// TIA Portal V20 export
// export: Created 2025-12-01T14:57:10.8516778Z, ExportSetting None, DisplayName Totally Integrated Automation Portal, DisplayVersion V20 Update 3, DisplayName TIA Portal Openness, DisplayVersion V20 Update 3, DisplayName TIA Portal Version Control Interface, DisplayVersion V20 Update 3, DisplayName STEP 7 Professional, DisplayVersion V20 Update 3, DisplayName STEP 7 Safety, DisplayVersion V20 Update 2, DisplayName WinCC Basic/Comfort/Advanced, DisplayVersion V20 Update 3, DisplayName WinCC Professional, DisplayVersion V20 Update 3, DisplayName WinCC Unified, DisplayVersion V20 Update 3
FUNCTION "FC823_OrdenesMesas" : Void   // FC823, LAD
TITLE = "OrdenesMesas" - Calcular las ordenes de las UT's
{ S7_Optimized_Access := 'FALSE' }
AUTHOR : TRACKING
NAME : 20160407
VERSION : 4.1
// - Inicializaciones
// - Bucle de Mesas
// - Cierre del Protocolo de la Mesa 
// - Buscar Nueva Orden para enviar a la Mesa
// - Calacular la nueva Orden de la Mesa
// stored: AutoNumber false, SetENOAutomatically false
   VAR_TEMP
      RecProtocoloDeMesa : "UDT_ProtocoloRecMesa";
      P_RecProtocolo : DWord;
      P_Temporal : DWord;
      PLCOrden : Word;   // Estructura de recepcion de la mesa
      PLCOrdenAux_01 : UInt;   // Estructura de recepcion de la mesa (TipoCarga)
      PLCMesaSalidaMultiple : UInt;   // Estructura de recepcion de la mesa (Auxiliar 02)
      PLCOrdenAux_03 : UInt;   // Estructura de recepcion de la mesa (Auxiliar 03)
      PLCOrdenAux_04 : UInt;   // Estructura de recepcion de la mesa (Auxiliar 04)
      NumeroMesa : UInt;   // Numero de Mesa Actual
      NumeroUT : UInt;   // Numero de UT Actual
      SiguienteUT : UInt;   // Numero de UT Siguiente
      ValorReturn : Int;   // Temporal
   END_VAR
BEGIN

NETWORK
TITLE = Inicializar
// Inicializacion de las variables de los DB's
/////////////////////////////////////////////////////////////////////////
// Inicializaciones de las variables de los DB's

      L     0;
      T     #PLCOrden;
      T     #PLCMesaSalidaMultiple;
      T     #PLCOrdenAux_01;
      T     #PLCOrdenAux_03;
      T     #PLCOrdenAux_04;



NETWORK
TITLE = Bucle de Mesas
// - Inicializacion de variables de la mesa (PunteroMesa y PunteroPLC)
// - Mirar si ha cerrado el protocolo
/////////////////////////////////////////////////////////////////////////
/////////////////////////////////////////////////////////////////////////
/////////////////////////////////////////////////////////////////////////
// Inicializo variable, para bucle de mesas
      L     0;
      T     #NumeroMesa;


/////////////////////////////////////////////////////////////////////////
// Inicializo variable, para bucle de mesas
// Empieza el recorrido por todas las Mesas
InicioBucle_Mesas:NOP   0;
      L     #NumeroMesa;  // Incremento en uno el numero de mesa
      L     1;
      +I;
      T     #NumeroMesa;


/////////////////////////////////////////////////////////////////////////
// Ya he recorrido todas las Mesas
      L     #NumeroMesa;  // Ya estan todas las Mesas
      L     "CTE_MaxMesas";
      >I;
      JC    _END;


/////////////////////////////////////////////////////////////////////////
/// Mirar Si hay Mesa Configurada, No Definida no seguir
      SET;
      AN    "DB850_DefinicionMesas".Mesa[#NumeroMesa].ConfigMesa.MesaPaso;
      AN    "DB850_DefinicionMesas".Mesa[#NumeroMesa].ConfigMesa.MesaCruce;
      AN    "DB850_DefinicionMesas".Mesa[#NumeroMesa].ConfigMesa.MesaMultiplesDestinos;
      AN    "DB850_DefinicionMesas".Mesa[#NumeroMesa].ConfigMesa.MesaTL;
      JC    InicioBucle_Mesas;


/////////////////////////////////////////////////////////////////////////
/// Recoger Datos de Emision y Recepcion
      CALL  MOVE
      ( IN  := "DB841_Recepcion".Mesa[#NumeroMesa].Protocolo,
        OUT := #RecProtocoloDeMesa
      );

      L     P##RecProtocoloDeMesa;
      T     #P_RecProtocolo;

/////////////////////////////////////////////////////////////////////////
// Mirar si ha cerrado el protocolo de la Mesa de la anterior orden enviada

// --- 1º Condicion: Tiene que estar cerrado el protocolo
      L     "DB810_ColasMesas".Colas[#NumeroMesa].EstadoOrdenMesa;
      L     0;  // Mirar si no esta Cerrado el Protocolo
      <>I;  // Ir a Cerrar Protocolo de la Mesa
      JC    CerrarProtocolo_Mesa;


/////////////////////////////////////////////////////////////////////////
// Ir a Buscar Orden Nueva para la Mesa
      JU    TratarOrden_Mesa;



NETWORK
TITLE = Cierre del protocolo de la mesa
// - Recoger como esta el RecepOK
// - Distribuir dependiendo del Status del Protocolo
// - Esta en Fase 1 - Esperando que se desactive RecepOK de la Mesa
// - Esta en Fase 2 - Esperando que se active RecepOK de la Mesa
CerrarProtocolo_Mesa:NOP   0;

/////////////////////////////////////////////////////////////////////////
/////////////////////////////////////////////////////////////////////////
/////////////////////////////////////////////////////////////////////////
/////////////////////////////////////////////////////////////////////////
// Distribuir dependiendo del Status del protocolo

      L     "DB810_ColasMesas".Colas[#NumeroMesa].EstadoOrdenMesa;
      L     1;  // Protocolo - Esta en Fase 1
      ==I;
      JC    ProtocoloEnFase_01_Mesa;

// Protocolo - Esta en Fase 2
      JU    ProtocoloEnFase_02_Mesa;


/////////////////////////////////////////////////////////////////////////
/////////////////////////////////////////////////////////////////////////
// Esta en Fase 1 - Esperando que se desactive RecepOK de la Mesa
ProtocoloEnFase_01_Mesa:NOP   0;
      SET;  // Si esta 1 todavia no se puede dar pòr finalizado el protocolo
      A     "DB840_Emision".Mesa[#NumeroMesa].Protocolo.RecepOK;
      JC    FinCerrarProtocolo_Mesa;

// Pasar a Fase 0, Acabado el Protocolo
      L     0;  // Fase 0
      T     "DB810_ColasMesas".Colas[#NumeroMesa].EstadoOrdenMesa;

      JU    FinCerrarProtocolo_Mesa;


/////////////////////////////////////////////////////////////////////////
/////////////////////////////////////////////////////////////////////////
// Esta en Fase 2 - Esperando que se active RecepOK de la Mesa
ProtocoloEnFase_02_Mesa:NOP   0;
      SET;  // Si esta a 0 todavia no cambia a fase 1 el protocolo
      AN    "DB840_Emision".Mesa[#NumeroMesa].Protocolo.RecepOK;
      JC    FinCerrarProtocolo_Mesa;

// Pasar a Fase 1, Esperando que desactive el RecpOK
      L     LW [#P_RecProtocolo];
      L     W#16#80;  // Desactivo la Orden enviada todas menos el bit EmiOK
      AW;  // Y todos los Word Adicionales se ponen a 0
      T     LW [#P_RecProtocolo];  // Posicion - 8

      CALL  MOVE
      ( IN  := #RecProtocoloDeMesa,
        OUT := "DB841_Recepcion".Mesa[#NumeroMesa].Protocolo
      );

      L     0;  // Word Auxiliares
      T     "DB841_Recepcion".Mesa[#NumeroMesa].MesaSalidaMultiDestino;
      T     "DB841_Recepcion".Mesa[#NumeroMesa].Auxiliar_01;
      T     "DB841_Recepcion".Mesa[#NumeroMesa].Auxiliar_03;
      T     "DB841_Recepcion".Mesa[#NumeroMesa].Auxiliar_04;

      L     1;  // Fase 1
      T     "DB810_ColasMesas".Colas[#NumeroMesa].EstadoOrdenMesa;

      JU    FinCerrarProtocolo_Mesa;


/////////////////////////////////////////////////////////////////////////
/////////////////////////////////////////////////////////////////////////
// Final del Segmento del Cierre de Protocolo de la Mesa
FinCerrarProtocolo_Mesa:NOP   0;
// Finalizar, ir a la siguiente Mesa
      JU    InicioBucle_Mesas;



NETWORK
TITLE = Buscar Nueva Orden a enviar al PLC (Solo la primera UT)
// - Mirar is hay UT (Solo tiene que enviar la primera de cada mesa)
// - Mirar como esta el VI (Estado)
// - Mirar si esta todo Emitido
// - Mirar si ha cambiado de Mesa
// - Mirar si ha recibido Evento
TratarOrden_Mesa:NOP   0;
      L     0;
      T     #PLCOrden;
      T     #PLCMesaSalidaMultiple;
      T     #PLCOrdenAux_01;
      T     #PLCOrdenAux_03;
      T     #PLCOrdenAux_04;

/////////////////////////////////////////////////////////////////////////
/////////////////////////////////////////////////////////////////////////
/////////////////////////////////////////////////////////////////////////
      L     "DB810_ColasMesas".Colas[#NumeroMesa].UT_PrimeraMesa;
      T     #NumeroUT;

/////////////////////////////////////////////////////////////////////////
// --- Mirar si hay UT, Si hay Inicializo el Puntero
// --- 1º Condicion: Tiene que haber UT en la Mesa

      L     #NumeroUT;  // Mirar si hay UT ?
      L     0;
      ==I;  // No hay UT
      JC    FinTratarOrden_Mesa;


/////////////////////////////////////////////////////////////////////////
// --- 2º Condicion: El estado del VI  ¡¡¡ ANALIZAR !!!
// ---   ¿Mirar como esta el VI?
// ---   ¿Solo cuando esta en Carga o reposo?
// ---   ¿Da lo mismo, menos en Reset?


/////////////////////////////////////////////////////////////////////////
// --- 3º Condicion: Estado del Dispositivo
// --- Condición >>> Marcha + Auto (EmisionDeDispositivoMesa)
// Marcha + Auto >> Sino esta asi NO puede Calcular la orden
      SET;
      A     "DB840_Emision".DispoMesa[#NumeroMesa].Protocolo.Automatico;
      A     "DB840_Emision".DispoMesa[#NumeroMesa].Protocolo.Marcha;
      JCN   FinTratarOrden_Mesa;


/////////////////////////////////////////////////////////////////////////
// --- Mirar si esta todo Emitido (StatusEmisionUT = 0)
// --- 4º Condicion: La UT no tiene nada Evento que Generar
//                   (Lo logico es que este libre, menos en un reset)
      L     "DB812_UTs_Control".UT[#NumeroUT].EstadoEmisionUT;
      L     0;
      <>I;  // Esta emitido todo ?
      JC    FinTratarOrden_Mesa;


/////////////////////////////////////////////////////////////////////////
/////////////////////////////////////////////////////////////////////////
/////////////////////////////////////////////////////////////////////////
// --- Mirar Si ha cambiado de estado (StatatusRecepcionUT <> 0)
// --- 1º Caso para el Calculo de Orden: Nueva UT ó Cambia Mesa
      L     "DB812_UTs_Control".UT[#NumeroUT].EstadoRecepcionUT;
      L     0;
      <>I;  // Si tiene para enviar orden ?
      JC    CalcularOrden_FASE01_Mesa;


/////////////////////////////////////////////////////////////////////////
/////////////////////////////////////////////////////////////////////////
/////////////////////////////////////////////////////////////////////////
// --- Mirar si ha Recibido Eventos (StatatusEventoRecibido <> 0)
// --- 2º Caso para el Calculo de Orden: Evento Recibido
// --- (Hay eventos que no tienen)
      L     "DB812_UTs_Control".UT[#NumeroUT].EstadoEventoRecibido;
      L     0;
      <>I;  // Si ha recibido Evento ?
      JC    RecibidoEvento_Mesa;


/////////////////////////////////////////////////////////////////////////
/////////////////////////////////////////////////////////////////////////
/////////////////////////////////////////////////////////////////////////
// No esta, no se puede enviar nada
      JU    FinTratarOrden_Mesa;


/////////////////////////////////////////////////////////////////////////
/////////////////////////////////////////////////////////////////////////
/////////////////////////////////////////////////////////////////////////
// Final del Segmento de Buscar Nueva Orden a enviar al PLC
FinTratarOrden_Mesa:NOP   0;
// Finalizar, ir a la siguiente Mesa
      JU    InicioBucle_Mesas;



NETWORK
TITLE = Recibido Evento para la Mesa
// - Distribucion dependiendo del ento recibido
// - Eventos que no necesitan Orden
//     - Recibido Evento de Borrar UT
//     - Recibido Evento de Refresco de datos la UT
// 
// -Eventos que puede ser que necesite orden
//     - Recibido Evento de Ruta Nueva
//     - Recibido Evento de Nueva UT Creada
//     - Recibido Evento de Nuevos Datos para la UT
//     - Recibido Evento de Retirar la UT
RecibidoEvento_Mesa:NOP   0;

/////////////////////////////////////////////////////////////////////////
/////////////////////////////////////////////////////////////////////////
/////////////////////////////////////////////////////////////////////////
// Distribucion de los Eventos Recibidos

      L     "DB812_UTs_Control".UT[#NumeroUT].EstadoEventoRecibido;
      L     201;  // 201 - Ruta Nueva
      ==I;
      JC    EventoRecido_RutaNuevaUT_Mesa;

      L     "DB812_UTs_Control".UT[#NumeroUT].EstadoEventoRecibido;
      L     202;  // 202 - UT Creada
      ==I;
      JC    EventoRecido_CreadaUT_Mesa;

      L     "DB812_UTs_Control".UT[#NumeroUT].EstadoEventoRecibido;
      L     203;  // 203 - BorrarUT
      ==I;
      JC    EventoRecido_BorrarUT_Mesa;

      L     "DB812_UTs_Control".UT[#NumeroUT].EstadoEventoRecibido;
      L     204;  // 204 - Datos Nuevos de la UT
      ==I;
      JC    EventoRecido_DatosNuevosUT_Mesa;

      L     "DB812_UTs_Control".UT[#NumeroUT].EstadoEventoRecibido;
      L     205;  // 205 - Referesco de Datos
      ==I;
      JC    EventoRecido_RefrescoDatosUT_Mesa;


/////////////////////////////////////////////////////////////////////////
// --- Solo queda este tipo de evento: Retirar UT
      L     "DB812_UTs_Control".UT[#NumeroUT].EstadoEventoRecibido;
      L     210;  // 210...214 - Retirar UT
      <I;  // < 210 ? - No es Retirar UT
      JC    NoRecibidoEvento_Retirar_Mesa;
      L     "DB812_UTs_Control".UT[#NumeroUT].EstadoEventoRecibido;
      L     214;  // 210...214 - Retirar UT
      >I;  // > 214 ? - No es Retirar UT
      JC    NoRecibidoEvento_Retirar_Mesa;

      SET;  // Si es orden de Retirar UT (Simple)
      AN    "DB850_DefinicionMesas".Mesa[#NumeroMesa].ConfigMesa.AusenciaMultiple;
      JC    EventoRecido_RetiradaSimpleUT_Mesa;

// Si es orden de Retirar UT (Multiple)
      JU    EventoRecido_RetiradaMultipleUT_Mesa;

NoRecibidoEvento_Retirar_Mesa:NOP   0;


/////////////////////////////////////////////////////////////////////////
// --- El evento recibido no lo espera el sistema  ¡¡¡ MALO, MALO, MALO !!!

      L     0;  // Dar por tratado el Evento
      L     "DB812_UTs_Control".UT[#NumeroUT].EstadoEventoRecibido;


// Fin del Tratamiento del Eventos
      JU    FinRecibidoEvento_Mesa;


/////////////////////////////////////////////////////////////////////////
/////////////////////////////////////////////////////////////////////////
/////////////////////////////////////////////////////////////////////////
/////////////////////////////////////////////////////////////////////////
// --- Final de tratamiento de los Eventos Recibidos
FinRecibidoEvento_Mesa:NOP   0;
// Finalizar, ir a la siguiente Mesa
      JU    InicioBucle_Mesas;



NETWORK
TITLE = --- Lista de Eventos Recibidos
/////////////////////////////////////////////////////////////////////////
/////////////////////////////////////////////////////////////////////////
/////////////////////////////////////////////////////////////////////////
//
//                  LISTA DE EVENTOS QUE SE PUEDEN RECIBIR
//                        QUE HACER EN CADA CASO
//
/////////////////////////////////////////////////////////////////////////
/////////////////////////////////////////////////////////////////////////
/////////////////////////////////////////////////////////////////////////


/////////////////////////////////////////////////////////////////////////
/////////////////////////////////////////////////////////////////////////
// --- Evento que no necesita Orden
// 203 --- Recibido Evento de Borrar _UT
EventoRecido_BorrarUT_Mesa:NOP   0;
      L     "DB812_UTs_Control".UT[#NumeroUT].EstadoGeneralUT;
      L     0;  // Si EstadoGeneralUT = 0
      <>I;  // Esta Libre ?
      JC    FinRecibidoEvento_Mesa;


// Continuar con el ciclo
      L     0;  // Dar por tratado el Evento
      T     "DB812_UTs_Control".UT[#NumeroUT].EstadoEventoRecibido;
      L     31;  // 31 - Peticion de Borrado de UT
      T     "DB812_UTs_Control".UT[#NumeroUT].EstadoGeneralUT;


// Fin del Tratamiento del Evento
      JU    FinRecibidoEvento_Mesa;


/////////////////////////////////////////////////////////////////////////
/////////////////////////////////////////////////////////////////////////
// --- Evento que no necesita Orden
// 205 --- Recibido Evento de Refresco de Datos de la UT
EventoRecido_RefrescoDatosUT_Mesa:NOP   0;
      L     "DB812_UTs_Control".UT[#NumeroUT].EstadoGeneralUT;  // EstadoGeneralUT = 0
      L     0;
      <>I;
      JC    FinRecibidoEvento_Mesa;  // Esta Libre ?


// Continuar con el ciclo
      L     0;  // Dar por tratado el Evento
      T     "DB812_UTs_Control".UT[#NumeroUT].EstadoEventoRecibido;
      L     22;  // 22 - Peticion de Refresco de datos
      T     "DB812_UTs_Control".UT[#NumeroUT].EstadoGeneralUT;


// Fin del Tratamiento del Evento
      JU    FinRecibidoEvento_Mesa;




/////////////////////////////////////////////////////////////////////////
/////////////////////////////////////////////////////////////////////////
/////////////////////////////////////////////////////////////////////////
/////////////////////////////////////////////////////////////////////////
// --- Evento que puede ser que necesite Orden
// 201 --- Recibido Evento de Ruta Nueva
EventoRecido_RutaNuevaUT_Mesa:NOP   0;
      L     0;  // Dar por tratado el Evento
      T     "DB812_UTs_Control".UT[#NumeroUT].EstadoEventoRecibido;
      L     17;  // 17 - Ruta Nueva
      T     "DB812_UTs_Control".UT[#NumeroUT].EstadoRecepcionUT;


// Ir a calcular la Nueva Orden
      JU    CalcularOrden_FASE01_Mesa;


/////////////////////////////////////////////////////////////////////////
/////////////////////////////////////////////////////////////////////////
// --- Evento que puede ser que necesite Orden
// 202 --- Recibido Evento de Nueva UT Creada
EventoRecido_CreadaUT_Mesa:NOP   0;
      L     0;  // Dar por tratado el Evento
      T     "DB812_UTs_Control".UT[#NumeroUT].EstadoEventoRecibido;
      L     16;  // 16 - UT Creada
      T     "DB812_UTs_Control".UT[#NumeroUT].EstadoRecepcionUT;


// Ir a calcular la Nueva Orden
      JU    CalcularOrden_FASE01_Mesa;


/////////////////////////////////////////////////////////////////////////
/////////////////////////////////////////////////////////////////////////
// --- Evento que puede ser que necesite Orden
// 204 --- Recibido Evento de Nuevos datos de la UT
EventoRecido_DatosNuevosUT_Mesa:NOP   0;
      L     0;  // Dar por tratado el Evento
      T     "DB812_UTs_Control".UT[#NumeroUT].EstadoEventoRecibido;
      L     15;  // 15 - Nuevos Datos de UT
      T     "DB812_UTs_Control".UT[#NumeroUT].EstadoRecepcionUT;


// Ir a calcular la Nueva Orden
      JU    CalcularOrden_FASE01_Mesa;



NETWORK
TITLE = --- Evento Recibido de Retirada (Control Especial)
/////////////////////////////////////////////////////////////////////////
/////////////////////////////////////////////////////////////////////////
// --- Evento que puede ser que necesite Orden (Simple)
// 210... 214 --- Recibido Evento de Retirar UT de la mesa
EventoRecido_RetiradaSimpleUT_Mesa:NOP   0;

// Activar Bit Recibido del Evento
      L     P##PLCOrden;  // Dirección de la Orden del PLC
      T     #P_Temporal;

      L     "DB812_UTs_Control".UT[#NumeroUT].EstadoEventoRecibido;
      L     210;
      -I;  // Numero de Bit a Activar
      L     #P_Temporal;
      +D;
      T     #P_Temporal;  // Direccion del Bit a Activar

      SET;  // Poner a '1' el bit de la orden
      S     L [#P_Temporal];  // Orden del PLC calculada


// Finalizar Evento Recibido
      L     0;  // Dar por tratado el Evento
      T     "DB812_UTs_Control".UT[#NumeroUT].EstadoEventoRecibido;


/////////////////////////////////////////////////////////////////////////
// Enviar la Orden al PLC
      JU    EnviarOrden_Al_PLC;




/////////////////////////////////////////////////////////////////////////
/////////////////////////////////////////////////////////////////////////
// --- Evento que puede ser que necesite Orden (Multiple)
// 210... 214 --- Recibido Evento de Retirar UT de la mesa
EventoRecido_RetiradaMultipleUT_Mesa:NOP   0;

      L     "DB812_UTs_Control".UT[#NumeroUT].UT_SiguienteMesa;
      T     #SiguienteUT;

/////////////////////////////////////////////////////////////////////////
// --- Primero Mirar si ha llegado la orden de Retirar a todas las UT's
InicioBucleVerificar_RetiradaMultipleUT_Mesa:NOP   0;
      L     #SiguienteUT;
      L     0;  // No hay más UT's
      ==I;  // No hay más UT's enviar Retirar
      JC    FinBucleVerificar_RetiradaMultipleUT_Mesa;

// EventoRecibido de la Primera UT == Evento Recibido de todas las UTs
      L     "DB812_UTs_Control".UT[#SiguienteUT].EstadoEventoRecibido;
      L     "DB812_UTs_Control".UT[#NumeroUT].EstadoEventoRecibido;
      <>I;  // Tienen que ser iguales todas las UTs
      JC    FinRecibidoEvento_Mesa;

// Recorrer todas las UT's
      L     "DB812_UTs_Control".UT[#SiguienteUT].UT_SiguienteMesa;
      T     #SiguienteUT;

      JU    InicioBucleVerificar_RetiradaMultipleUT_Mesa;

// Final de Veficacion, Todas las Uts tienen Retirada
FinBucleVerificar_RetiradaMultipleUT_Mesa:NOP   0;


/////////////////////////////////////////////////////////////////////////
// Activar Bit Recibido del Evento
      L     P##PLCOrden;  // Dirección de la Orden del PLC
      T     #P_Temporal;

      L     "DB812_UTs_Control".UT[#NumeroUT].EstadoEventoRecibido;
      L     210;
      -I;  // Numero de Bit a Activar
      L     #P_Temporal;
      +D;
      T     #P_Temporal;  // Direccion del Bit a Activar

      SET;  // Poner a '1' el bit de la orden
      S     L [#P_Temporal];  // Orden del PLC calculada


/////////////////////////////////////////////////////////////////////////
// Dar por tratado el Evento Recibido Primera UT
      L     0;  // Dar por tratado el Evento
      T     "DB812_UTs_Control".UT[#NumeroUT].EstadoEventoRecibido;


/////////////////////////////////////////////////////////////////////////
// Dar por tratado el Evento Recibido al Resto de UT's
      L     "DB812_UTs_Control".UT[#NumeroUT].UT_SiguienteMesa;
      T     #SiguienteUT;

InicioBucleTratado_RetiradaMultipleUT_Mesa:NOP   0;
      L     #SiguienteUT;
      L     0;  // No hay más UT's
      ==I;  // No hay más UT's Finalizado
      JC    FinBucleTratado_RetiradaMultipleUT_Mesa;

// Dar por tratado el Evento
      L     0;  // Dar por tratado el Evento
      T     "DB812_UTs_Control".UT[#SiguienteUT].EstadoEventoRecibido;

// Recorrer todas las UT's
      L     "DB812_UTs_Control".UT[#SiguienteUT].UT_SiguienteMesa;
      T     #SiguienteUT;

      JU    InicioBucleTratado_RetiradaMultipleUT_Mesa;

// Final de Tratado, Todas las Uts tienen tratado el Evenfo
FinBucleTratado_RetiradaMultipleUT_Mesa:NOP   0;


/////////////////////////////////////////////////////////////////////////
/////////////////////////////////////////////////////////////////////////
// Enviar la Orden al PLC
      JU    EnviarOrden_Al_PLC;




NETWORK
TITLE = Calcular Orden - FASE 01 (Distribucion Causa) ---- Nota >>> Primera UT de la Mesa
CalcularOrden_FASE01_Mesa:NOP   0;

/////////////////////////////////////////////////////////////////////////
/////////////////////////////////////////////////////////////////////////
/////////////////////////////////////////////////////////////////////////
// Distribucion segun la causa:

      L     "DB812_UTs_Control".UT[#NumeroUT].EstadoRecepcionUT;
      L     11;  //  - (11) : Cambiado de Mesa la UT
      ==I;
      JC    CambiadaDeMesa_CalcularOrden_Mesa;

      L     "DB812_UTs_Control".UT[#NumeroUT].EstadoRecepcionUT;
      L     12;  //  - (12) : Nueva UT en Mesa
      ==I;
      JC    NuevaEnMesa_CalcularOrden_Mesa;

      L     "DB812_UTs_Control".UT[#NumeroUT].EstadoRecepcionUT;
      L     13;  //  - (13) : Reset del PLC
      ==I;
      JC    ResetEnMesa_CalcularOrden_Mesa;

      L     "DB812_UTs_Control".UT[#NumeroUT].EstadoRecepcionUT;
      L     15;  //  - (15) : Datos Nuevos de la UT
      ==I;
      JC    DatosNuevos_CalcularOrden_Mesa;

      L     "DB812_UTs_Control".UT[#NumeroUT].EstadoRecepcionUT;
      L     16;  //  - (16) : Creada UT
      ==I;
      JC    CreadaEnMesa_CalcularOrden_Mesa;

      L     "DB812_UTs_Control".UT[#NumeroUT].EstadoRecepcionUT;
      L     17;  //  - (17) : Recibida Nueva Ruta para la UT
      ==I;
      JC    RutaNueva_CalcularOrden_Mesa;


/////////////////////////////////////////////////////////////////////////
// --- No es una causa programada (Darla por tradada)
      L     0;  // Dar por tratada
      T     "DB812_UTs_Control".UT[#NumeroUT].EstadoRecepcionUT;

// No hay más que hacer
      JU    InicioBucle_Mesas;



NETWORK
TITLE = --- EstadoRecepcion (11) : Cambiado de Mesa la UT
// Pasos a Seguir: 
// - Mirar condiciones que debe cumplir
// - Calcular la Orden a Enviar
// - Darla por tratada y enviar la orden si es necesario
CambiadaDeMesa_CalcularOrden_Mesa:NOP   0;

/////////////////////////////////////////////////////////////////////////
/////////////////////////////////////////////////////////////////////////
/////////////////////////////////////////////////////////////////////////
// (11) : Cambiado de Mesa la UT


/////////////////////////////////////////////////////////////////////////
// --- Mirar condiciones que debe cumplir


/////////////////////////////////////////////////////////////////////////
// --- Calcular Orden
      JU    CalcularOrden_FASE02_Mesa;



NETWORK
TITLE = --- EstadoRecepcion (12) : Nueva UT en Mesa
// Pasos a Seguir: 
// - Mirar condiciones que debe cumplir
// - Calcular la Orden a Enviar
// - Darla por tratada y enviar la orden si es necesario
NuevaEnMesa_CalcularOrden_Mesa:NOP   0;

/////////////////////////////////////////////////////////////////////////
/////////////////////////////////////////////////////////////////////////
/////////////////////////////////////////////////////////////////////////
// (12) : Nueva UT en Mesa


/////////////////////////////////////////////////////////////////////////
// --- Mirar condiciones que debe cumplir


/////////////////////////////////////////////////////////////////////////
// --- Se da la causa por tratata, no se envia orden
      L     0;  // Dar por tratada
      T     "DB812_UTs_Control".UT[#NumeroUT].EstadoRecepcionUT;

// No hay más que hacer
      JU    InicioBucle_Mesas;



NETWORK
TITLE = --- EstadoRecepcion (13) : Reset de la UT
// Pasos a Seguir: 
// - Mirar condiciones que debe cumplir
// - Calcular la Orden a Enviar
// - Darla por tratada y enviar la orden si es necesario
ResetEnMesa_CalcularOrden_Mesa:NOP   0;

/////////////////////////////////////////////////////////////////////////
/////////////////////////////////////////////////////////////////////////
/////////////////////////////////////////////////////////////////////////
// (13) : Reset de la UT

/////////////////////////////////////////////////////////////////////////
// --- Mirar condiciones que debe cumplir


/////////////////////////////////////////////////////////////////////////
// --- Calcular Orden
      JU    CalcularOrden_FASE02_Mesa;



NETWORK
TITLE = --- EstadoRecepcion (15) : Datos Nuevos de la UT
// Pasos a Seguir: 
// - Mirar condiciones que debe cumplir
// - Calcular la Orden a Enviar
// - Darla por tratada y enviar la orden si es necesario
DatosNuevos_CalcularOrden_Mesa:NOP   0;

/////////////////////////////////////////////////////////////////////////
/////////////////////////////////////////////////////////////////////////
/////////////////////////////////////////////////////////////////////////
// (15) : Datos Nuevos de la UT


/////////////////////////////////////////////////////////////////////////
// --- Mirar condiciones que debe cumplir


/////////////////////////////////////////////////////////////////////////
// --- Se da la causa por tratata, no se envia orden
      L     0;  // Dar por tratada
      T     "DB812_UTs_Control".UT[#NumeroUT].EstadoRecepcionUT;

// No hay más que hacer
      JU    InicioBucle_Mesas;



NETWORK
TITLE = --- EstadoRecepcion (16) : Creada UT
// Pasos a Seguir: 
// - Mirar condiciones que debe cumplir
// - Calcular la Orden a Enviar
// - Darla por tratada y enviar la orden si es necesario
CreadaEnMesa_CalcularOrden_Mesa:NOP   0;

/////////////////////////////////////////////////////////////////////////
/////////////////////////////////////////////////////////////////////////
/////////////////////////////////////////////////////////////////////////
// (16) : Creada UT


/////////////////////////////////////////////////////////////////////////
// --- Mirar condiciones que debe cumplir


/////////////////////////////////////////////////////////////////////////
// --- Se da la causa por tratata, no se envia orden
      L     0;  // Dar por tratada
      T     "DB812_UTs_Control".UT[#NumeroUT].EstadoRecepcionUT;

// No hay más que hacer
      JU    InicioBucle_Mesas;



NETWORK
TITLE = --- EstadoRecepcion (17) : Recibida Nueva Ruta para la UT
// Pasos a Seguir: 
// - Mirar condiciones que debe cumplir
// - Calcular la Orden a Enviar
// - Darla por tratada y enviar la orden si es necesario
RutaNueva_CalcularOrden_Mesa:NOP   0;

/////////////////////////////////////////////////////////////////////////
/////////////////////////////////////////////////////////////////////////
/////////////////////////////////////////////////////////////////////////
// (17) : Recibida Nueva Ruta para la UT


/////////////////////////////////////////////////////////////////////////
// --- Mirar condiciones que debe cumplir


/////////////////////////////////////////////////////////////////////////
// --- Calcular Orden
      JU    CalcularOrden_FASE02_Mesa;



NETWORK
TITLE = Calcular Orden - FASE 02 (Control Comun de la UT)
CalcularOrden_FASE02_Mesa:NOP   0;

/////////////////////////////////////////////////////////////////////////
/////////////////////////////////////////////////////////////////////////
/////////////////////////////////////////////////////////////////////////
//                    OPERATIVA NORMAL DE FUNCIONAMIENTO
/////////////////////////////////////////////////////////////////////////
// Casos que se puede dar:
//
// 1 Si no tiene Mckey, No debe darse este caso, tenerlo previsto.
//   Realizar, Evento de Nueva UT en Mesa (NUNCA SE DARA)
// 2 Sino tiene Ruta, MesaDestino = 0 (NUNCA SE DARA)
//   Realizar, Evento de Pedir Nueva Ruta
// 3 Si tiene ruta y ha llegado a su destino
// 4 Si tiene ruta y no ha llegado a su destino
//
/////////////////////////////////////////////////////////////////////////


/////////////////////////////////////////////////////////////////////////
// --- 1º Caso: El Mckey = 0 (Evento de Nueva UT en Mesa)
/////////////////////////////////////////////////////////////////////////
// El McKey = 0 (Evento de Nueva UT en la Mesa)
// Este caso NUNCA se dará, pero se programa por si acaso.
      SET;
      L     "DB812_UTs_Control".UT[#NumeroUT].Mckey;
      L     0;
      ==D;  // Tiene Mckey ?
      JC    NoEsxiteMckey_CalcularOrden_Mesa;


/////////////////////////////////////////////////////////////////////////
// --- 2º Caso: No tiene Ruta (MesaDestino = 0) (Evento de Pedir Ruta)
/////////////////////////////////////////////////////////////////////////
// El MesaDestino = 0 (Evento de Pedir Ruta Nueva)
// Este caso NUNCA se dará, pero se programa por si acaso.

      SET;  // Memoria de Recibido la Orden RETI (Prioritario)
      A     "DB812_UTs_Control".UT[#NumeroUT].AtributosDeLaUT.MemorizarRETI;
      JC    MemorizadoRetirada_CalcularOrden_Mesa;

      L     "DB812_UTs_Control".UT[#NumeroUT].MesaDestino;
      L     0;  // No tiene destino
      ==I;  // Tiene Ruta ?
      JC    SinDestino_CalcularOrden_Mesa;


/////////////////////////////////////////////////////////////////////////
// --- 3º Caso: Hay Ruta, y ha llegado a su destino (MesaDestino = MesaActual)
// --- MODIFICACION 06/05/2013 --> Recircular Activado, debe dar una vuelta completa
// ---       Aunque ha llegado su Destino, si esta activado la Marca
// ---       debe recircular siempre.

      SET;  // Memoria de Recibido la Orden RETI (Prioritario)
      A     "DB812_UTs_Control".UT[#NumeroUT].AtributosDeLaUT.MemorizarRETI;
      JC    MemorizadoRetirada_CalcularOrden_Mesa;

      SET;  // Solo para mesas de Cruce, Debe Recicular
      A     "DB812_UTs_Control".UT[#NumeroUT].AtributosDeLaUT.RecircularCarga;
      A     "DB850_DefinicionMesas".Mesa[#NumeroMesa].ConfigMesa.MesaCruce;
      JC    NoComprobarDestino_CalcularOrden_Mesa;

      L     "DB812_UTs_Control".UT[#NumeroUT].MesaDestino;
      L     "DB812_UTs_Control".UT[#NumeroUT].MesaActual;
      ==I;  // Ha llegado a su Destino ?
      JC    EnDestino_CalcularOrden_Mesa;

// Fin de Control de Llegada a Destino
NoComprobarDestino_CalcularOrden_Mesa:NOP   0;


/////////////////////////////////////////////////////////////////////////
// --- 4º Caso: Hay Ruta, y no ha llegado a su destino (MesaDestino <> MesaActual)
//     La UT esta de camino a su destino, dependiendo del tipo de mesa


/////////////////////////////////////////////////////////////////////////
// --- Si Bit de la Definicion de la Mesa "EspecialOrdenes", Hay funcion especial
//     que calcula la orden a enviar

      SET;
      A     "DB850_DefinicionMesas".Mesa[#NumeroMesa].ConfigMesa.EspecialOrdenes;  // Hay funcion particular
      JC    InicioBucle_Mesas;  // Aqui no hay nada que hacer


/////////////////////////////////////////////////////////////////////////
// --- Hay que hacer cosas diferentes, dependiendo del Tipo de Mesa:
//     * Mesa tipo de PASO
//     * Mesa tipo de CRUCE
//     * Mesa tipo de MUTIPLES DESTINOS
//     * Si no hay definido >>> No se Hace Nada

      SET;  // Es una Mesa de Paso
      A     "DB850_DefinicionMesas".Mesa[#NumeroMesa].ConfigMesa.MesaPaso;
      JC    MesaDePaso_CalcularOrden_Mesa;

      SET;  // Es una Mesa de Cruce
      A     "DB850_DefinicionMesas".Mesa[#NumeroMesa].ConfigMesa.MesaCruce;
      JC    MesaDeCruce_CalcularOrden_Mesa;

      SET;  // Es una Mesa de Multiples Destinos
      A     "DB850_DefinicionMesas".Mesa[#NumeroMesa].ConfigMesa.MesaMultiplesDestinos;
      JC    MesaDeMultiplesDestinos_CalcularOrden_Mesa;


/////////////////////////////////////////////////////////////////////////
// Tienen que estar la MESA configurada
      JU    InicioBucle_Mesas;



NETWORK
TITLE = --- Control (CASO) : No Tiene Mckey
NoEsxiteMckey_CalcularOrden_Mesa:NOP   0;

/////////////////////////////////////////////////////////////////////////
/////////////////////////////////////////////////////////////////////////
/////////////////////////////////////////////////////////////////////////
/////////////////////////////////////////////////////////////////////////
// --- El Mckey = 0 (Evento de Nueva UT en Mesa)
/////////////////////////////////////////////////////////////////////////
// El McKey = 0 (Evento de Nueva UT en la Mesa)
// Este caso NUNCA se dará, pero se programa por si acaso.


/////////////////////////////////////////////////////////////////////////
// Condiciones -- EstadoGeneralUT = 0
      L     "DB812_UTs_Control".UT[#NumeroUT].EstadoGeneralUT;
      L     0;  // Libre
      <>I;  // NO esta LIBRE ?
      JC    InicioBucle_Mesas;


/////////////////////////////////////////////////////////////////////////
// Acciones:   -- EstadoGeneralUT = 24 (Evento de Nueva UT en Mesa)
//             -- EstadoRecepcionUT = 0
      L     24;  // 24 - Generar Evento Nueva UT en Mesa
      T     "DB812_UTs_Control".UT[#NumeroUT].EstadoGeneralUT;
      L     0;  // Dar por tratada
      T     "DB812_UTs_Control".UT[#NumeroUT].EstadoRecepcionUT;

// No hay más que hacer
      JU    InicioBucle_Mesas;



NETWORK
TITLE = --- Control (CASO) : No tiene Destino
SinDestino_CalcularOrden_Mesa:NOP   0;

/////////////////////////////////////////////////////////////////////////
/////////////////////////////////////////////////////////////////////////
/////////////////////////////////////////////////////////////////////////
/////////////////////////////////////////////////////////////////////////
// --- No tiene Ruta (MesaDestino = 0) (Evento de Pedir Ruta)
/////////////////////////////////////////////////////////////////////////
// El MesaDestino = 0 (Evento de Pedir Ruta Nueva)
// Este caso NUNCA se dará, pero se programa por si acaso.


/////////////////////////////////////////////////////////////////////////
// Condiciones -- EstadoGeneralUT = 0
      L     "DB812_UTs_Control".UT[#NumeroUT].EstadoGeneralUT;
      L     0;  // Libre
      <>I;  // NO esta LIBRE ?
      JC    InicioBucle_Mesas;


/////////////////////////////////////////////////////////////////////////
// Acciones:   -- EstadoGeneralUT = 25 (Evento de Pedir Ruta Nueva)
//             -- EstadoRecepcionUT = 0
      L     25;  // 25 - Generar Evento Pedir Ruta (SIN DESTINO)
      T     "DB812_UTs_Control".UT[#NumeroUT].EstadoGeneralUT;
      L     0;  // Dar por tratada
      T     "DB812_UTs_Control".UT[#NumeroUT].EstadoRecepcionUT;

// No hay más que hacer
      JU    InicioBucle_Mesas;



NETWORK
TITLE = --- Control (CASO) : En Destino
EnDestino_CalcularOrden_Mesa:NOP   0;

/////////////////////////////////////////////////////////////////////////
/////////////////////////////////////////////////////////////////////////
/////////////////////////////////////////////////////////////////////////
/////////////////////////////////////////////////////////////////////////
// --- Ha llegado a su desetino (Evento de Pedir Ruta)
/////////////////////////////////////////////////////////////////////////
// MesaActual = MesaDestino(Evento de Pedir Ruta Nueva)


/////////////////////////////////////////////////////////////////////////
// Condiciones -- EstadoGeneralUT = 0
      L     "DB812_UTs_Control".UT[#NumeroUT].EstadoGeneralUT;
      L     0;  // Libre
      <>I;  // NO esta LIBRE ?
      JC    InicioBucle_Mesas;


/////////////////////////////////////////////////////////////////////////
// Acciones:   -- EstadoGeneralUT = 21 (Evento de Pedir Ruta Nueva)
//             -- EstadoRecepcionUT = 0
      L     21;  // 21 - Generar Evento Pedir Ruta
      T     "DB812_UTs_Control".UT[#NumeroUT].EstadoGeneralUT;
      L     0;  // Dar por tratada
      T     "DB812_UTs_Control".UT[#NumeroUT].EstadoRecepcionUT;

// No hay más que hacer
      JU    InicioBucle_Mesas;



NETWORK
TITLE = --- Control (CASO) : Memorizado Evento de Retirada
MemorizadoRetirada_CalcularOrden_Mesa:NOP   0;

/////////////////////////////////////////////////////////////////////////
/////////////////////////////////////////////////////////////////////////
/////////////////////////////////////////////////////////////////////////
/////////////////////////////////////////////////////////////////////////
// --- Esta activado el RETI
//     SE MEMORIZA SALIDA EN MESA INTERMEDIA (21 03 2016)
//     EstadoEventoRecibido = Mesa Intermeria (Salida RETI)

      L     "DB812_UTs_Control".UT[#NumeroUT].MesaIntermedia;
      T     "DB812_UTs_Control".UT[#NumeroUT].EstadoEventoRecibido;
      L     0;  // Dar por tratada
      T     "DB812_UTs_Control".UT[#NumeroUT].EstadoRecepcionUT;

// No hay más que hacer
      JU    InicioBucle_Mesas;



NETWORK
TITLE = Calcular Orden - FASE Final >>> Mesa De Paso
MesaDePaso_CalcularOrden_Mesa:NOP   0;

/////////////////////////////////////////////////////////////////////////
/////////////////////////////////////////////////////////////////////////
/////////////////////////////////////////////////////////////////////////
/////////////////////////////////////////////////////////////////////////
//  Calcular Orden para MESA de PASO

      CALL  "FC825_CalcularOrdenUT_MesaPaso"
      ( NumeroUT        := #NumeroUT,
        Orden           := #PLCOrden,
        Auxiliar_01     := #PLCOrdenAux_01,
        MesaSalidaMulti := #PLCMesaSalidaMultiple,
        Auxiliar_03     := #PLCOrdenAux_03,
        Auxiliar_04     := #PLCOrdenAux_04
      );


/////////////////////////////////////////////////////////////////////////
// Enviar la Orden al PLC
      JU    EnviarOrden_Al_PLC;



NETWORK
TITLE = Calcular Orden - FASE Final >>> Mesa De Cruce
MesaDeCruce_CalcularOrden_Mesa:NOP   0;

/////////////////////////////////////////////////////////////////////////
/////////////////////////////////////////////////////////////////////////
/////////////////////////////////////////////////////////////////////////
/////////////////////////////////////////////////////////////////////////
//  Calcular Orden para MESA de CRUCE

      CALL  "FC826_CalcularOrdenUT_MesaCruce"
      ( NumeroUT        := #NumeroUT,
        Orden           := #PLCOrden,
        Auxiliar_01     := #PLCOrdenAux_01,
        MesaSalidaMulti := #PLCMesaSalidaMultiple,
        Auxiliar_03     := #PLCOrdenAux_03,
        Auxiliar_04     := #PLCOrdenAux_04
      );


/////////////////////////////////////////////////////////////////////////
// Enviar la Orden al PLC
      JU    EnviarOrden_Al_PLC;



NETWORK
TITLE = Calcular Orden - FASE Final >>> Mesa De Multiples Destinos
MesaDeMultiplesDestinos_CalcularOrden_Mesa:NOP   0;

/////////////////////////////////////////////////////////////////////////
/////////////////////////////////////////////////////////////////////////
/////////////////////////////////////////////////////////////////////////
/////////////////////////////////////////////////////////////////////////
//  Calcular Orden para MESA de MULTIPLES DESTINOS

      CALL  "FC827_CalcularOrdenUT_MesaMultiDestino"
      ( NumeroUT        := #NumeroUT,
        Orden           := #PLCOrden,
        Auxiliar_01     := #PLCOrdenAux_01,
        MesaSalidaMulti := #PLCMesaSalidaMultiple,
        Auxiliar_03     := #PLCOrdenAux_03,
        Auxiliar_04     := #PLCOrdenAux_04
      );


/////////////////////////////////////////////////////////////////////////
// Enviar la Orden al PLC
      JU    EnviarOrden_Al_PLC;



NETWORK
TITLE = Enviar la Orden al PLC
EnviarOrden_Al_PLC:NOP   0;

/////////////////////////////////////////////////////////////////////////
/////////////////////////////////////////////////////////////////////////
/////////////////////////////////////////////////////////////////////////
// --- Enviar orden si la hay
      L     #PLCOrden;  // Mirar si hay orden para enviar
      L     0;
      ==I;  // No hay Orden para enviar?
      JC    FinEnviarOrden_Al_PLC;


/////////////////////////////////////////////////////////////////////////
// --- Hay orden, enviarla

      L     LW [#P_RecProtocolo];  // Bits de Recepcion de la Mesa
      L     #PLCOrden;  // Activo la Nueva Orden
      OW;
      T     LW [#P_RecProtocolo];  // Bits de Recepcion de la Mesa

      CALL  MOVE
      ( IN  := #RecProtocoloDeMesa,
        OUT := "DB841_Recepcion".Mesa[#NumeroMesa].Protocolo
      );

      L     #PLCOrdenAux_01;
      T     "DB841_Recepcion".Mesa[#NumeroMesa].Auxiliar_01;
      L     #PLCMesaSalidaMultiple;
      T     "DB841_Recepcion".Mesa[#NumeroMesa].MesaSalidaMultiDestino;
      L     #PLCOrdenAux_03;
      T     "DB841_Recepcion".Mesa[#NumeroMesa].Auxiliar_03;
      L     #PLCOrdenAux_04;
      T     "DB841_Recepcion".Mesa[#NumeroMesa].Auxiliar_04;


// Pasar a Fase 2, Esperando que active el RecpOK
      L     2;  // Fase 2
      T     "DB810_ColasMesas".Colas[#NumeroMesa].EstadoOrdenMesa;

      JU    FinEnviarOrden_Al_PLC;




/////////////////////////////////////////////////////////////////////////
/////////////////////////////////////////////////////////////////////////
/////////////////////////////////////////////////////////////////////////
// Final del Segmento de Buscar Nueva Orden a enviar al PLC
FinEnviarOrden_Al_PLC:NOP   0;
// Finalizar, ir a la siguiente mesa
      JU    InicioBucle_Mesas;



NETWORK
TITLE = Final
// Se acabo la funcion
_END: NOP   0;

END_FUNCTION
